// Mitsubishi GX Works2 project: LRI - PLC - SELO COM RESET   PLC: Q03UDV

PROGRAM MAIN
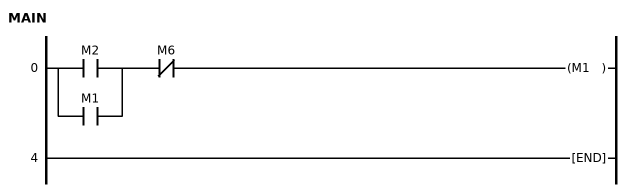
0     LD      M2
      OR      M1
      ANI     M6
      OUT     M1
4     END
END_PROGRAM
